// TwinCAT 3 PLC project Plc
// ProgramVersion: 3.1.4024.0
// libraries:
//   Tc2_MC2, * (Beckhoff Automation GmbH)
//   Tc2_Standard, * (Beckhoff Automation GmbH)
//   Tc2_System, * (Beckhoff Automation GmbH)
//   Tc3_Module, * (Beckhoff Automation GmbH)
//   VisuSymbols,3.5.10.0,System
// project tree:
//   / Gestore di visualizzazione.TcVMO (not stored), GlobalTextList.TcGTLO, PlcTask.TcTTO
//   GVLs/ GVL.TcGVL
//   POUs/ MAIN.TcPOU
//   VISUs/ Visualization.TcVIS
// real-time tasks:
//   TASK PlcTask: cycle T#10ms, priority 20, ADS port 350
// motion (NC):
//   TASK NC-Task 1 SAF: cycle T#2ms, priority 4, ADS port 501
//   TASK NC-Task 1 SVB: cycle T#10ms, priority 8, ADS port 511
//   AXIS Asse virtuale (id 1)
//     OtherSettings: AllowMotionCmdToSlave=true
//     encoder EncType=1
//     drive DrvType=5
//       Analog: TorqueSetpointScale=10, ScaleFactorActTorque=0.1
//       TimeComp: TaskDelayCycles=1
//     controller CtrType=1
//       CtrPara: PriorControlFactor=1
//         Observer: BandWidth=20
// variable links:
//   Plc/Plc Instance <-> NC-Task 1 SAF/Axes/Asse virtuale
//     PlcTask Inputs/GVL.axis.NcToPlc <-> Outputs/ToPlc
//     PlcTask Outputs/GVL.axis.PlcToNc <-> Inputs/FromPlc

CONFIGURATION Plc
    RESOURCE PLC ON TwinCAT3
        TASK PlcTask(INTERVAL := T#10ms, PRIORITY := 20);
        PROGRAM MAIN WITH PlcTask : MAIN;
    END_RESOURCE
END_CONFIGURATION

// ---- GVLs/GVL.TcGVL
{attribute 'qualified_only'}
VAR_GLOBAL
	Axis: AXIS_REF;
	pAbilitaMotore: BOOL;
	pDisabilitaMotore: BOOL;
	motoreAbilitato: BOOL;
	pAbilitaJog: BOOL;
	bErrorJog: BOOL;
	pMoveVelocity: BOOL;
	pHalt: BOOL;
END_VAR

// ---- POUs/MAIN.TcPOU
PROGRAM MAIN
VAR
	MCPower: MC_Power;
	McJog: MC_Jog;
	McReadStatus: MC_ReadStatus;
	McMoveVelocity: MC_MoveVelocity;
	McHalt: MC_Halt;
END_VAR

EnableAxis();
Jog();
MoveVelocity();
Halt();
ReadStatus();

ACTION EnableAxis:
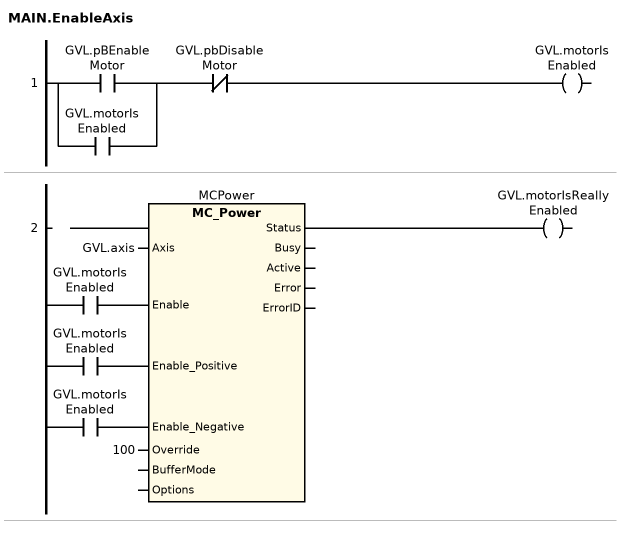
// NETWORK 1
GVL.motorIsEnabled := (GVL.pBEnableMotor OR GVL.motorIsEnabled) AND NOT GVL.pbDisableMotor;

// NETWORK 2
MCPower(
    Axis := GVL.axis,
    Enable := GVL.motorIsEnabled,
    Enable_Positive := GVL.motorIsEnabled,
    Enable_Negative := GVL.motorIsEnabled,
    Override := 100); // MC_Power
GVL.motorIsReallyEnabled := MCPower.Status;
END_ACTION

ACTION Halt:
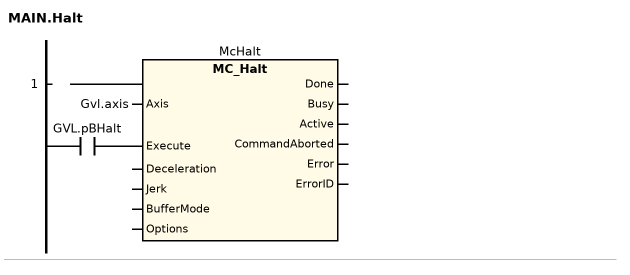
// NETWORK 1
McHalt(Axis := Gvl.axis, Execute := GVL.pBHalt); // MC_Halt
END_ACTION

ACTION Jog:
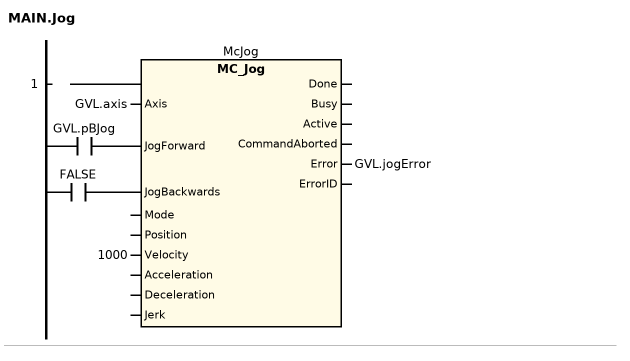
// NETWORK 1
McJog(
    Axis := GVL.axis,
    JogForward := GVL.pBJog,
    JogBackwards := FALSE,
    Velocity := 1000,
    Error => GVL.jogError); // MC_Jog
END_ACTION

ACTION MoveVelocity:
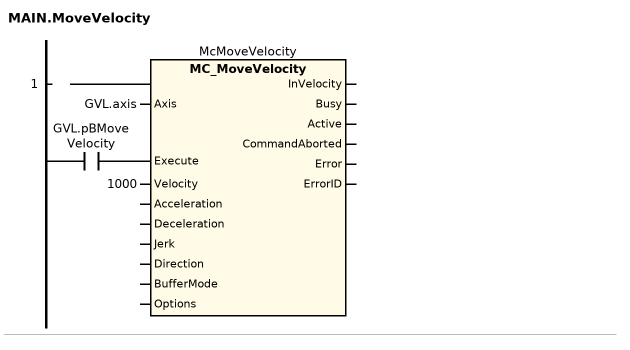
// NETWORK 1
McMoveVelocity(Axis := GVL.axis, Execute := GVL.pBMoveVelocity, Velocity := 1000); // MC_MoveVelocity
END_ACTION

ACTION ReadStatus:
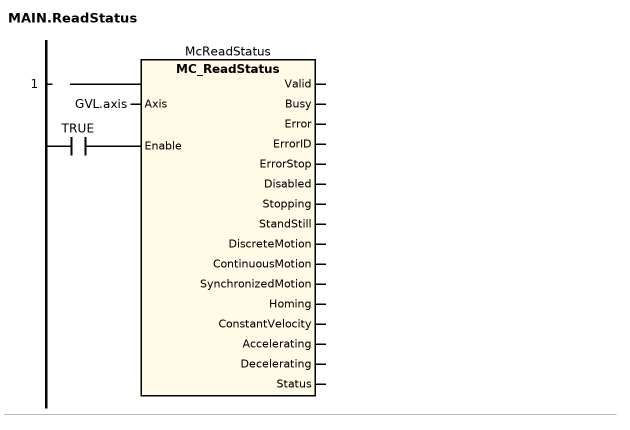
// NETWORK 1
McReadStatus(Axis := GVL.axis, Enable := TRUE); // MC_ReadStatus
END_ACTION

END_PROGRAM

// ---- GlobalTextList.TcGTLO
TEXTLIST GlobalTextList
  4 = '%d'
  166 = 'Abilita motore'
  310 = 'Disabilita motore'
  622 = 'Errore Jog'
  426 = 'Errore motore'
  859 = 'Halt'
  5 = 'Jog'
  351 = 'Motore abilitato'
  664 = 'Motore in movimento'
  831 = 'Move Velocity'
  104 = 'Posizione motore'
  227 = 'Testo'
END_TEXTLIST

// ---- VISUs/Visualization.TcVIS
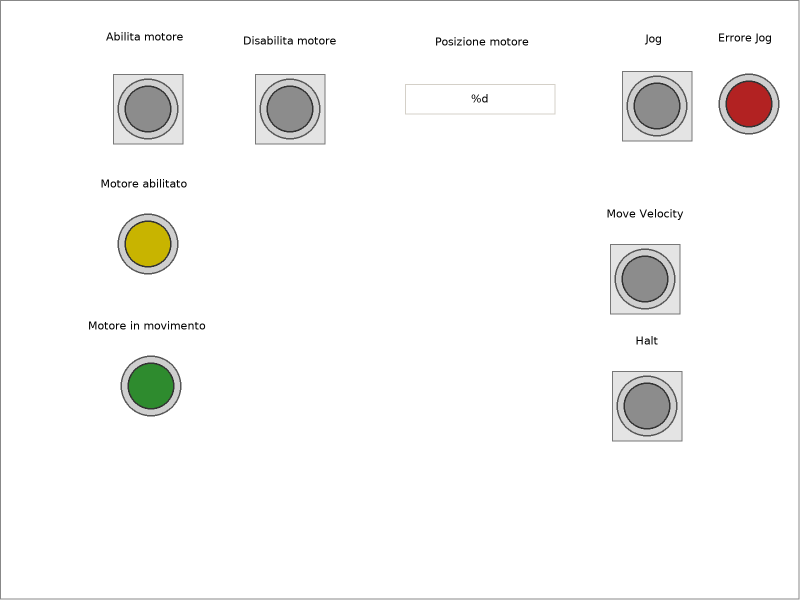
VISUALIZATION Visualization  // 800x600
    PushSwitch (113,74 70x70), variable: GVL.pAbilitaMotore, behaviour: TAP, style: Switch-PushSwitch-Gray
    Lamp1 (113,209 70x70), variable: GVL.motoreAbilitato, style: Lamp-Lamp1-Yellow
    Label (69,169 150x30), "Motore abilitato"
    Label (70,22 150x30), "Abilita motore"
    PushSwitch (255,74 70x70), variable: GVL.pDisabilitaMotore, behaviour: TAP, style: Switch-PushSwitch-Gray
    Label (215,26 150x30), "Disabilita motore"
    Textfield (405,84 150x30), "%d", text variable: GVL.Axis.NcToPlc.ActPos
    PushSwitch (622,71 70x70), variable: GVL.pAbilitaJog, behaviour: TAP, style: Switch-PushSwitch-Gray
    Label (579,24 150x30), "Jog"
    Lamp1 (116,351 70x70), variable: GVL.Axis.Status.Moving, style: Lamp-Lamp1-Green
    Label (72,311 150x30), "Motore in movimento"
    Lamp1 (714,69 70x70), variable: GVL.bErrorJog, style: Lamp-Lamp1-Red
    Label (670,23 150x30), "Errore Jog"
    Label (407,27 150x30), "Posizione motore"
    PushSwitch (610,244 70x70), variable: GVL.pMoveVelocity, behaviour: TAP, style: Switch-PushSwitch-Gray
    Label (570,199 150x30), "Move Velocity"
    PushSwitch (612,371 70x70), variable: GVL.pHalt, behaviour: TAP, style: Switch-PushSwitch-Gray
    Label (572,326 150x30), "Halt"
END_VISUALIZATION
